# EPICS substitutions: apps/Alias4527App/Db/SY4527_crate14.substitutions
# Provide a reset signal.
# This doesn't actually do anything because the SY4527 doesn't have a way
# to reset via EPICS.  So it provides a No-op for the GUI to attach to.
# Peraps a future firmware for the SY4527 will have a reset signal, or we can
# rig up an output register to send a reset signal.
file "db/Reset4527.template" {
pattern
     {P,     H}
     {hchv, 14}
}
# Slot 0
file db/SY4527_readbacks.template {
    pattern { P, H, S, V}
        { hchv, 14, 00, 000}
        { hchv, 14, 00, 001}
        { hchv, 14, 00, 002}
        { hchv, 14, 00, 003}
        { hchv, 14, 00, 004}
        { hchv, 14, 00, 005}
        { hchv, 14, 00, 006}
        { hchv, 14, 00, 007}
        { hchv, 14, 00, 008}
        { hchv, 14, 00, 009}
        { hchv, 14, 00, 010}
        { hchv, 14, 00, 011}
        { hchv, 14, 00, 012}
        { hchv, 14, 00, 013}
        { hchv, 14, 00, 014}
        { hchv, 14, 00, 015}
        { hchv, 14, 00, 016}
        { hchv, 14, 00, 017}
        { hchv, 14, 00, 018}
        { hchv, 14, 00, 019}
        { hchv, 14, 00, 020}
        { hchv, 14, 00, 021}
        { hchv, 14, 00, 022}
        { hchv, 14, 00, 023}
}
# Slot 2
file db/SY4527_readbacks.template {
    pattern { P, H, S, V}
        { hchv, 14, 02, 000}
        { hchv, 14, 02, 001}
        { hchv, 14, 02, 002}
        { hchv, 14, 02, 003}
        { hchv, 14, 02, 004}
        { hchv, 14, 02, 005}
        { hchv, 14, 02, 006}
        { hchv, 14, 02, 007}
        { hchv, 14, 02, 008}
        { hchv, 14, 02, 009}
        { hchv, 14, 02, 010}
        { hchv, 14, 02, 011}
        { hchv, 14, 02, 012}
        { hchv, 14, 02, 013}
        { hchv, 14, 02, 014}
        { hchv, 14, 02, 015}
        { hchv, 14, 02, 016}
        { hchv, 14, 02, 017}
        { hchv, 14, 02, 018}
        { hchv, 14, 02, 019}
        { hchv, 14, 02, 020}
        { hchv, 14, 02, 021}
        { hchv, 14, 02, 022}
        { hchv, 14, 02, 023}
}
# Slot 4
file db/SY4527_readbacks.template {
    pattern { P, H, S, V}
        { hchv, 14, 04, 000}
        { hchv, 14, 04, 001}
        { hchv, 14, 04, 002}
        { hchv, 14, 04, 003}
        { hchv, 14, 04, 004}
        { hchv, 14, 04, 005}
        { hchv, 14, 04, 006}
        { hchv, 14, 04, 007}
        { hchv, 14, 04, 008}
        { hchv, 14, 04, 009}
        { hchv, 14, 04, 010}
        { hchv, 14, 04, 011}
        { hchv, 14, 04, 012}
        { hchv, 14, 04, 013}
        { hchv, 14, 04, 014}
        { hchv, 14, 04, 015}
        { hchv, 14, 04, 016}
        { hchv, 14, 04, 017}
        { hchv, 14, 04, 018}
        { hchv, 14, 04, 019}
        { hchv, 14, 04, 020}
        { hchv, 14, 04, 021}
        { hchv, 14, 04, 022}
        { hchv, 14, 04, 023}
}
# Slot 6
file db/SY4527_readbacks.template {
    pattern { P, H, S, V}
        { hchv, 14, 06, 000}
        { hchv, 14, 06, 001}
        { hchv, 14, 06, 002}
        { hchv, 14, 06, 003}
        { hchv, 14, 06, 004}
        { hchv, 14, 06, 005}
        { hchv, 14, 06, 006}
        { hchv, 14, 06, 007}
        { hchv, 14, 06, 008}
        { hchv, 14, 06, 009}
        { hchv, 14, 06, 010}
        { hchv, 14, 06, 011}
        { hchv, 14, 06, 012}
        { hchv, 14, 06, 013}
        { hchv, 14, 06, 014}
        { hchv, 14, 06, 015}
        { hchv, 14, 06, 016}
        { hchv, 14, 06, 017}
        { hchv, 14, 06, 018}
        { hchv, 14, 06, 019}
        { hchv, 14, 06, 020}
        { hchv, 14, 06, 021}
        { hchv, 14, 06, 022}
        { hchv, 14, 06, 023}
}
# Slot 8
file db/SY4527_readbacks.template {
    pattern { P, H, S, V}
        { hchv, 14, 08, 000}
        { hchv, 14, 08, 001}
        { hchv, 14, 08, 002}
        { hchv, 14, 08, 003}
        { hchv, 14, 08, 004}
        { hchv, 14, 08, 005}
        { hchv, 14, 08, 006}
        { hchv, 14, 08, 007}
        { hchv, 14, 08, 008}
        { hchv, 14, 08, 009}
        { hchv, 14, 08, 010}
        { hchv, 14, 08, 011}
        { hchv, 14, 08, 012}
        { hchv, 14, 08, 013}
        { hchv, 14, 08, 014}
        { hchv, 14, 08, 015}
        { hchv, 14, 08, 016}
        { hchv, 14, 08, 017}
        { hchv, 14, 08, 018}
        { hchv, 14, 08, 019}
        { hchv, 14, 08, 020}
        { hchv, 14, 08, 021}
        { hchv, 14, 08, 022}
        { hchv, 14, 08, 023}
}
# Slot 10
file db/SY4527_readbacks.template {
    pattern { P, H, S, V}
        { hchv, 14, 10, 000}
        { hchv, 14, 10, 001}
        { hchv, 14, 10, 002}
        { hchv, 14, 10, 003}
        { hchv, 14, 10, 004}
        { hchv, 14, 10, 005}
        { hchv, 14, 10, 006}
        { hchv, 14, 10, 007}
        { hchv, 14, 10, 008}
        { hchv, 14, 10, 009}
        { hchv, 14, 10, 010}
        { hchv, 14, 10, 011}
        { hchv, 14, 10, 012}
        { hchv, 14, 10, 013}
        { hchv, 14, 10, 014}
        { hchv, 14, 10, 015}
        { hchv, 14, 10, 016}
        { hchv, 14, 10, 017}
        { hchv, 14, 10, 018}
        { hchv, 14, 10, 019}
        { hchv, 14, 10, 020}
        { hchv, 14, 10, 021}
        { hchv, 14, 10, 022}
        { hchv, 14, 10, 023}
}
# Slot 12
file db/SY4527_readbacks.template {
    pattern { P, H, S, V}
        { hchv, 14, 12, 000}
        { hchv, 14, 12, 001}
        { hchv, 14, 12, 002}
        { hchv, 14, 12, 003}
        { hchv, 14, 12, 004}
        { hchv, 14, 12, 005}
        { hchv, 14, 12, 006}
        { hchv, 14, 12, 007}
        { hchv, 14, 12, 008}
        { hchv, 14, 12, 009}
        { hchv, 14, 12, 010}
        { hchv, 14, 12, 011}
        { hchv, 14, 12, 012}
        { hchv, 14, 12, 013}
        { hchv, 14, 12, 014}
        { hchv, 14, 12, 015}
        { hchv, 14, 12, 016}
        { hchv, 14, 12, 017}
        { hchv, 14, 12, 018}
        { hchv, 14, 12, 019}
        { hchv, 14, 12, 020}
        { hchv, 14, 12, 021}
        { hchv, 14, 12, 022}
        { hchv, 14, 12, 023}
}
# Slot 14
file db/SY4527_readbacks.template {
    pattern { P, H, S, V}
        { hchv, 14, 14, 000}
        { hchv, 14, 14, 001}
        { hchv, 14, 14, 002}
        { hchv, 14, 14, 003}
        { hchv, 14, 14, 004}
        { hchv, 14, 14, 005}
        { hchv, 14, 14, 006}
        { hchv, 14, 14, 007}
        { hchv, 14, 14, 008}
        { hchv, 14, 14, 009}
        { hchv, 14, 14, 010}
        { hchv, 14, 14, 011}
        { hchv, 14, 14, 012}
        { hchv, 14, 14, 013}
        { hchv, 14, 14, 014}
        { hchv, 14, 14, 015}
        { hchv, 14, 14, 016}
        { hchv, 14, 14, 017}
        { hchv, 14, 14, 018}
        { hchv, 14, 14, 019}
        { hchv, 14, 14, 020}
        { hchv, 14, 14, 021}
        { hchv, 14, 14, 022}
        { hchv, 14, 14, 023}
}
